SUBAPPLICATION Versuch_404 (* Versuch Array Summe *)
  (* Standard: 61499-2; Description: Copyright (c) 2023 Meisterschulen am Ostbahnhof This program and the accompanying materials are made available under the terms of the Eclipse Public License 2.0 which is available at https://www.eclipse.org/legal/epl-2.0/ SPDX-License-Identifier: EPL-2.0 *)
  (* Version 1.0, 2023-10-23, Franz Höpfinger, Meisterschulen am Ostbahnhof *)
  PACKAGE Versuche;
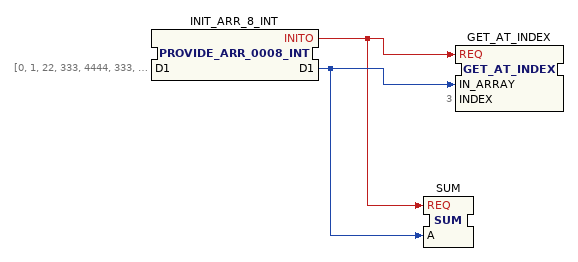
  FBS
    INIT_ARR_8_INT : eclipse4diac::convert::providers::PROVIDE_ARR_0008_INT(D1 := [0, 1, 22, 333, 4444, 333, 22, 1]);
    GET_AT_INDEX : eclipse4diac::convert::GET_AT_INDEX(INDEX := 3);
    SUM : logiBUS::utils::dyn_arr::SUM;
  END_FBS
  EVENT_CONNECTIONS
    INIT_ARR_8_INT.INITO TO GET_AT_INDEX.REQ;
    INIT_ARR_8_INT.INITO TO SUM.REQ;
  END_CONNECTIONS
  DATA_CONNECTIONS
    INIT_ARR_8_INT.D1 TO GET_AT_INDEX.IN_ARRAY;
    INIT_ARR_8_INT.D1 TO SUM.A;
  END_CONNECTIONS
END_SUBAPPLICATION
